{region '#Template'}
	{attribute 'Version' := '5.0.0.0'}
	{attribute 'Tags' := '"LCID": "1031", "Text": "Universal, Multistate, Aggregate"'}
	{attribute 'Tags' := '"LCID": "1033", "Text": "Universal, Multistate, Aggregate"'}
	{attribute 'Using' := '"Type": "Template", "URI": "EC_ID"'}
	{attribute 'Using' := '"Type": "Template", "URI": "BA2_Param"'}
	{attribute 'Description' := '"LCID": "1031", "Text": "Aktor multistate"'}
	{attribute 'Description' := '"LCID": "1033", "Text": "Actuator multistate"'}
{endregion}			 
FUNCTION_BLOCK FB_BA_ActuatorMultistate EXTENDS FB_BA_View
VAR_INPUT
	stCmd					: ST_BA_MultiState;	
END_VAR
VAR_OUTPUT
	nCmd					: UDINT;
	bDst					: BOOL;
	eActivePrio				: E_BA_Priority;
END_VAR
VAR_INPUT CONSTANT	
	Cmd						: FB_BA_MO_Raw;	
	PlantLock				: FB_BA_PlantLock;	
END_VAR
VAR
	bPrioSfty				: BOOL;
	bPrioCrit				: BOOL;	
END_VAR
VAR // added by the converter: edge detectors and wires of the graphical bodies
    _w1 : ANY;
END_VAR

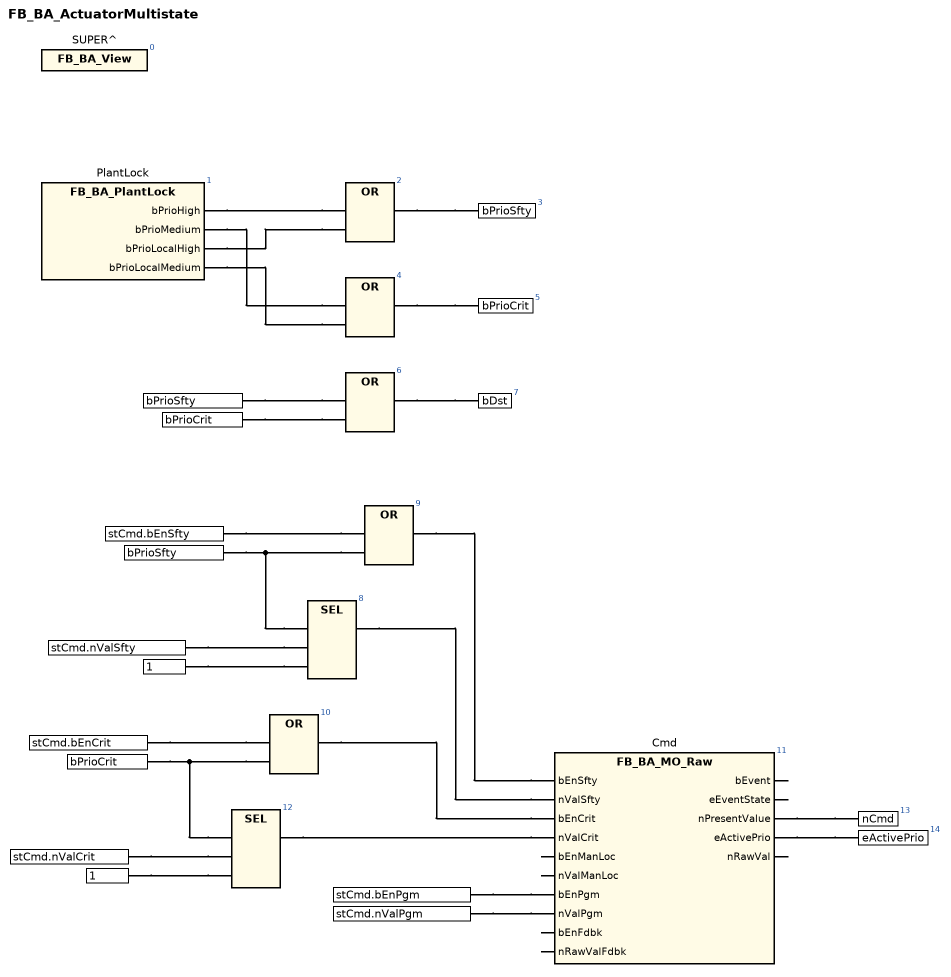
SUPER^(); // FB_BA_View
PlantLock(); // FB_BA_PlantLock
bPrioSfty := PlantLock.bPrioHigh OR PlantLock.bPrioLocalHigh;
bPrioCrit := PlantLock.bPrioMedium OR PlantLock.bPrioLocalMedium;
bDst := bPrioSfty OR bPrioCrit;
Cmd(
    bEnSfty := stCmd.bEnSfty OR bPrioSfty,
    nValSfty := SEL(bPrioSfty, stCmd.nValSfty, 1),
    bEnCrit := stCmd.bEnCrit OR bPrioCrit,
    nValCrit := _w1,
    bEnPgm := stCmd.bEnPgm,
    nValPgm := stCmd.nValPgm); // FB_BA_MO_Raw
_w1 := SEL(bPrioCrit, stCmd.nValCrit, 1);
nCmd := Cmd.nPresentValue;
eActivePrio := Cmd.eActivePrio;

METHOD FB_init : BOOL
VAR_INPUT
	bInitRetains : BOOL; // if TRUE, the retain variables are initialized (warm start / cold start)
	bInCopyCode : BOOL;  // if TRUE, the instance afterwards gets moved into the copy code (online change)
END_VAR
PlantLock.Parent				:= THIS^;	

Cmd.iParent						:= THIS^;
Cmd.iLabel						:= LblFun_SwitchingCommand;
Cmd.aStateText[1]				:= txtEvent_Stop;
Cmd.aStateText[2]				:= txtEvent_Open;
Cmd.aStateText[3]				:= txtEvent_Close;
Cmd.bEnManualRm					:= FALSE;	//	Priority  8	
Cmd.nValManualRm				:= 1;		//	Priority  8
Cmd.nDefaultValue				:= 1;	
Cmd.nEventClassID				:= EC_ID.NC80;
Cmd.stTimeDelay.nToNormal		:= BA2_Param.nDefTimeDelay_ToNormal;
Cmd.stTimeDelay.nToAbnormal		:= BA2_Param.nDefTimeDelay_ToAbnormal;
Cmd.aEventTransitionText[1]		:= txtEvent_Disturb;
Cmd.aEventTransitionText[2]		:= txtEvent_None;
Cmd.aEventTransitionText[3]		:= txtEvent_Normal;
Cmd.bEventDetectionEnable		:= FALSE;
Cmd.eEnPlantLock				:= E_BA_LockPriority.eNoLock;
END_METHOD

END_FUNCTION_BLOCK

(* stored: Version 1.1.0.1, ProductVersion 3.1.4024.12
   POU FB_BA_ActuatorMultistate: Id {6408e48a-1952-4833-8b14-0bc8352cde42}, SpecialFunc None
   Method FB_init: Id {d64aac7b-8976-47e6-97dd-ce25f7ddb26c} *)
